FUNCTION_BLOCK TOnTimer
VAR
    TON1 : TON;
END_VAR

METHOD Delay : BOOL
VAR_INPUT
    In : BOOL;
END_VAR
TON1(IN := In);
Delay := TON1.Q;
END_METHOD

METHOD FB_init : BOOL
VAR_INPUT
	bInitRetains : BOOL; // if TRUE, the retain variables are initialized (warm start / cold start)
	bInCopyCode : BOOL;  // if TRUE, the instance afterwards gets moved into the copy code (online change)
    PresetTime : LREAL; // seconds
END_VAR
TON1.PT := LREAL_TO_TIME(PresetTime * 1000);
END_METHOD

PROPERTY OutputState : BOOL
GET
OutputState := TON1.Q;
END_GET
END_PROPERTY

PROPERTY PresetTime : LREAL
GET
PresetTime := TIME_TO_LREAL(TON1.PT)/1000.0; // in seconds
END_GET
SET
TON1.PT := LREAL_TO_TIME(PresetTime * 1000);
END_SET
END_PROPERTY

METHOD Reset
TON1(IN := FALSE);
END_METHOD

METHOD Run : BOOL
TON1(IN := TRUE);
Run := TON1.Q;
END_METHOD

END_FUNCTION_BLOCK

(* stored: Version 1.1.0.1, ProductVersion 3.1.4024.3
   POU TOnTimer: Id {677fc192-31a0-06a7-0135-9ed2e1b8f627}, SpecialFunc None
   Method Delay: Id {0d9559ec-6c29-008c-30e1-2b6c5be571d9}
   Method FB_init: Id {523937ce-f181-060a-3975-d17e94bc8381}
   Property OutputState: Id {a28b64ed-1563-4b91-a7f3-215fbd1f41f8}
   Get Get: Id {b7210633-a708-400f-ae47-b4297bcc670f}
   Property PresetTime: Id {c5774100-9185-0102-0bda-dd487567e0a1}
   Get Get: Id {03d9bde0-ef32-06e4-3d0b-1ec1280df1ca}
   Set Set: Id {aec92e53-4db2-0128-3a07-41119aeed772}
   Method Reset: Id {ca2fbbd6-ed37-0717-0d86-2b0978515b06}
   Method Run: Id {74695f11-d12a-0d18-1144-977d6a8d3fd7} *)
